// TIA Portal V21 export
FUNCTION "ANALOG" : Void   // FC9, LAD
{ S7_Optimized_Access := 'TRUE' }
// stored: SetENOAutomatically false
   VAR_TEMP
      DOOR1_P : Real;
      DOOR2_P : Real;
      CHAMBER_P : Real;
      JACKET_P : Real;
      NOM : Real;
      TEMP1 : Real;
   END_VAR
   VAR_TEMP   // added for the SCL form of the ladder/FBD networks
      _w1 : Bool;
      _w2 : Bool;
      _w3 : Bool;
   END_VAR
BEGIN

REGION Network 1: TEMPERATURE RTD
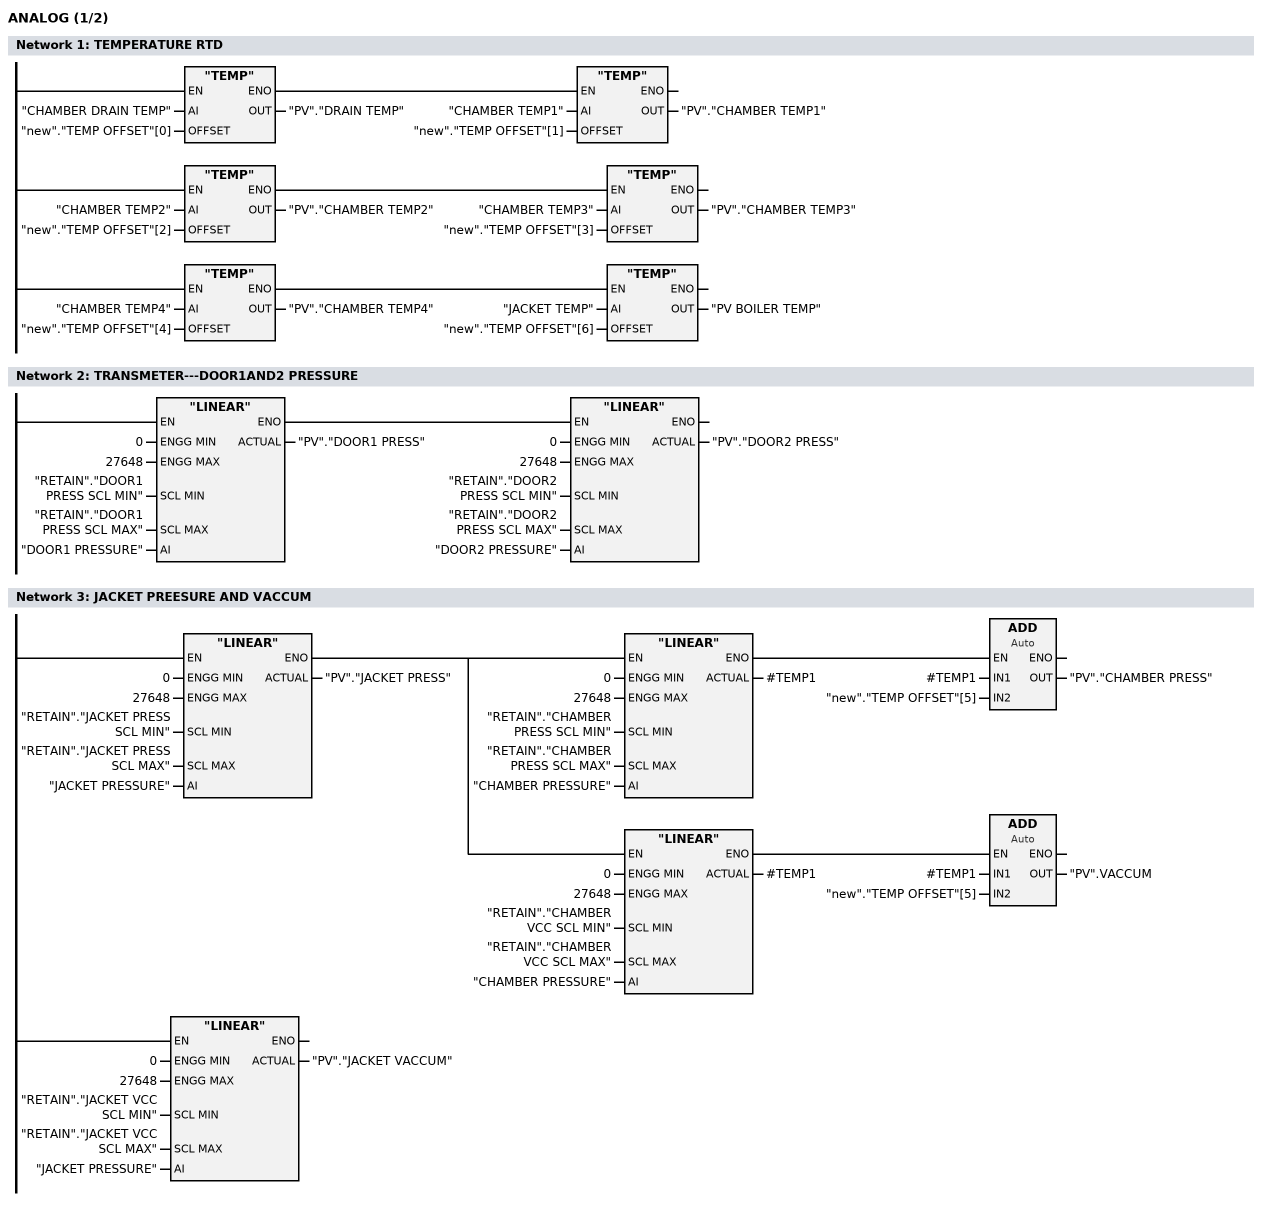
   RUNG wire#powerrail
      "TEMP"(AI := "CHAMBER DRAIN TEMP", OFFSET := "new"."TEMP OFFSET"[0], OUT => "PV"."DRAIN TEMP")
      "TEMP"(AI := "CHAMBER TEMP1", OFFSET := "new"."TEMP OFFSET"[1], OUT => "PV"."CHAMBER TEMP1")
   END_RUNG
   RUNG wire#powerrail
      "TEMP"(AI := "CHAMBER TEMP2", OFFSET := "new"."TEMP OFFSET"[2], OUT => "PV"."CHAMBER TEMP2")
      "TEMP"(AI := "CHAMBER TEMP3", OFFSET := "new"."TEMP OFFSET"[3], OUT => "PV"."CHAMBER TEMP3")
   END_RUNG
   RUNG wire#powerrail
      "TEMP"(AI := "CHAMBER TEMP4", OFFSET := "new"."TEMP OFFSET"[4], OUT => "PV"."CHAMBER TEMP4")
      "TEMP"(AI := "JACKET TEMP", OFFSET := "new"."TEMP OFFSET"[6], OUT => "PV BOILER TEMP")
   END_RUNG
   // the same network as SCL:
   "TEMP"(AI := "CHAMBER DRAIN TEMP", OFFSET := "new"."TEMP OFFSET"[0], OUT => "PV"."DRAIN TEMP", ENO => #_w1);
   IF #_w1 THEN
       "TEMP"(AI := "CHAMBER TEMP1", OFFSET := "new"."TEMP OFFSET"[1], OUT => "PV"."CHAMBER TEMP1");
   END_IF;
   "TEMP"(AI := "CHAMBER TEMP2", OFFSET := "new"."TEMP OFFSET"[2], OUT => "PV"."CHAMBER TEMP2", ENO => #_w2);
   IF #_w2 THEN
       "TEMP"(AI := "CHAMBER TEMP3", OFFSET := "new"."TEMP OFFSET"[3], OUT => "PV"."CHAMBER TEMP3");
   END_IF;
   "TEMP"(AI := "CHAMBER TEMP4", OFFSET := "new"."TEMP OFFSET"[4], OUT => "PV"."CHAMBER TEMP4", ENO => #_w3);
   IF #_w3 THEN
       "TEMP"(AI := "JACKET TEMP", OFFSET := "new"."TEMP OFFSET"[6], OUT => "PV BOILER TEMP");
   END_IF;
END_REGION

REGION Network 2: TRANSMETER---DOOR1AND2 PRESSURE
   RUNG wire#powerrail
      "LINEAR"("ENGG MIN" := 0, "ENGG MAX" := 27648, "SCL MIN" := "RETAIN"."DOOR1 PRESS SCL MIN", "SCL MAX" := "RETAIN"."DOOR1 PRESS SCL MAX", AI := "DOOR1 PRESSURE", ACTUAL => "PV"."DOOR1 PRESS")
      "LINEAR"("ENGG MIN" := 0, "ENGG MAX" := 27648, "SCL MIN" := "RETAIN"."DOOR2 PRESS SCL MIN", "SCL MAX" := "RETAIN"."DOOR2 PRESS SCL MAX", AI := "DOOR2 PRESSURE", ACTUAL => "PV"."DOOR2 PRESS")
   END_RUNG
   // the same network as SCL:
   "LINEAR"("ENGG MIN" := 0,
            "ENGG MAX" := 27648,
            "SCL MIN" := "RETAIN"."DOOR1 PRESS SCL MIN",
            "SCL MAX" := "RETAIN"."DOOR1 PRESS SCL MAX",
            AI := "DOOR1 PRESSURE",
            ACTUAL => "PV"."DOOR1 PRESS",
            ENO => #_w1);
   IF #_w1 THEN
       "LINEAR"("ENGG MIN" := 0,
                "ENGG MAX" := 27648,
                "SCL MIN" := "RETAIN"."DOOR2 PRESS SCL MIN",
                "SCL MAX" := "RETAIN"."DOOR2 PRESS SCL MAX",
                AI := "DOOR2 PRESSURE",
                ACTUAL => "PV"."DOOR2 PRESS");
   END_IF;
END_REGION

REGION Network 3: JACKET PREESURE AND VACCUM
   RUNG wire#powerrail
      "LINEAR"("ENGG MIN" := 0, "ENGG MAX" := 27648, "SCL MIN" := "RETAIN"."JACKET PRESS SCL MIN", "SCL MAX" := "RETAIN"."JACKET PRESS SCL MAX", AI := "JACKET PRESSURE", ACTUAL => "PV"."JACKET PRESS")
      wire#w1
      "LINEAR"("ENGG MIN" := 0, "ENGG MAX" := 27648, "SCL MIN" := "RETAIN"."CHAMBER PRESS SCL MIN", "SCL MAX" := "RETAIN"."CHAMBER PRESS SCL MAX", AI := "CHAMBER PRESSURE", ACTUAL => #TEMP1)
      Add(in1 := #TEMP1, in2 := "new"."TEMP OFFSET"[5], out => "PV"."CHAMBER PRESS")
   END_RUNG
   RUNG wire#w1
      "LINEAR"("ENGG MIN" := 0, "ENGG MAX" := 27648, "SCL MIN" := "RETAIN"."CHAMBER VCC SCL MIN", "SCL MAX" := "RETAIN"."CHAMBER VCC SCL MAX", AI := "CHAMBER PRESSURE", ACTUAL => #TEMP1)
      Add(in1 := #TEMP1, in2 := "new"."TEMP OFFSET"[5], out => "PV".VACCUM)
   END_RUNG
   RUNG wire#powerrail
      "LINEAR"("ENGG MIN" := 0, "ENGG MAX" := 27648, "SCL MIN" := "RETAIN"."JACKET VCC SCL MIN", "SCL MAX" := "RETAIN"."JACKET VCC SCL MAX", AI := "JACKET PRESSURE", ACTUAL => "PV"."JACKET VACCUM")
   END_RUNG
   // the same network as SCL:
   "LINEAR"("ENGG MIN" := 0,
            "ENGG MAX" := 27648,
            "SCL MIN" := "RETAIN"."JACKET PRESS SCL MIN",
            "SCL MAX" := "RETAIN"."JACKET PRESS SCL MAX",
            AI := "JACKET PRESSURE",
            ACTUAL => "PV"."JACKET PRESS",
            ENO => #_w1);
   "LINEAR"(EN := #_w1,
            "ENGG MIN" := 0,
            "ENGG MAX" := 27648,
            "SCL MIN" := "RETAIN"."CHAMBER PRESS SCL MIN",
            "SCL MAX" := "RETAIN"."CHAMBER PRESS SCL MAX",
            AI := "CHAMBER PRESSURE",
            ACTUAL => #TEMP1,
            ENO => #_w2);
   IF #_w2 THEN "PV"."CHAMBER PRESS" := #TEMP1 + "new"."TEMP OFFSET"[5]; END_IF;
   "LINEAR"(EN := #_w1,
            "ENGG MIN" := 0,
            "ENGG MAX" := 27648,
            "SCL MIN" := "RETAIN"."CHAMBER VCC SCL MIN",
            "SCL MAX" := "RETAIN"."CHAMBER VCC SCL MAX",
            AI := "CHAMBER PRESSURE",
            ACTUAL => #TEMP1,
            ENO => #_w3);
   IF #_w3 THEN "PV".VACCUM := #TEMP1 + "new"."TEMP OFFSET"[5]; END_IF;
   "LINEAR"("ENGG MIN" := 0,
            "ENGG MAX" := 27648,
            "SCL MIN" := "RETAIN"."JACKET VCC SCL MIN",
            "SCL MAX" := "RETAIN"."JACKET VCC SCL MAX",
            AI := "JACKET PRESSURE",
            ACTUAL => "PV"."JACKET VACCUM");
END_REGION

REGION Network 4: DOOR1AND 2 VACCUM
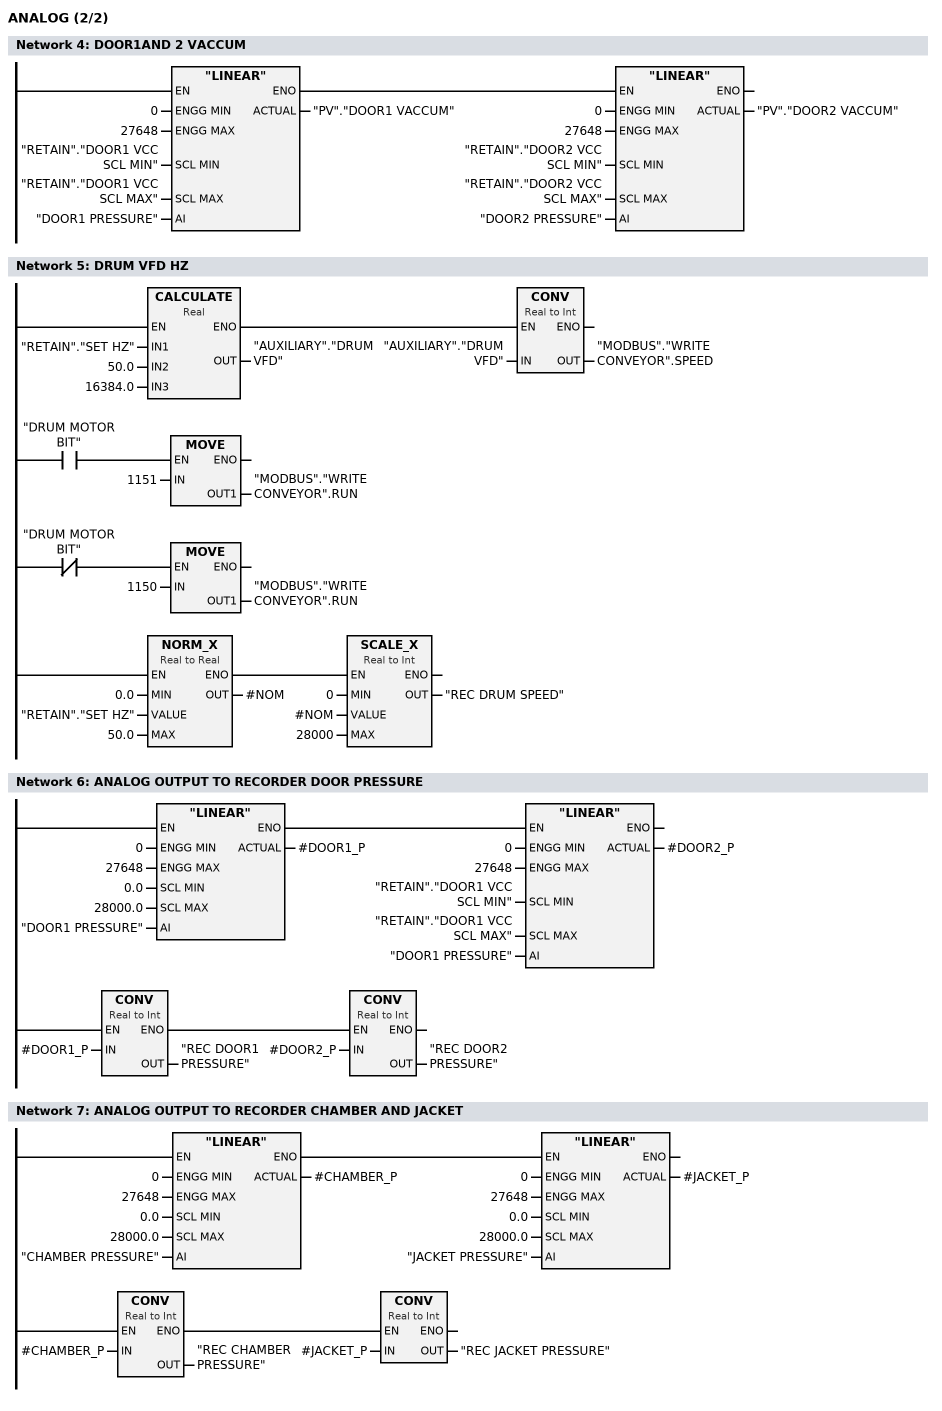
   RUNG wire#powerrail
      "LINEAR"("ENGG MIN" := 0, "ENGG MAX" := 27648, "SCL MIN" := "RETAIN"."DOOR1 VCC SCL MIN", "SCL MAX" := "RETAIN"."DOOR1 VCC SCL MAX", AI := "DOOR1 PRESSURE", ACTUAL => "PV"."DOOR1 VACCUM")
      "LINEAR"("ENGG MIN" := 0, "ENGG MAX" := 27648, "SCL MIN" := "RETAIN"."DOOR2 VCC SCL MIN", "SCL MAX" := "RETAIN"."DOOR2 VCC SCL MAX", AI := "DOOR2 PRESSURE", ACTUAL => "PV"."DOOR2 VACCUM")
   END_RUNG
   // the same network as SCL:
   "LINEAR"("ENGG MIN" := 0,
            "ENGG MAX" := 27648,
            "SCL MIN" := "RETAIN"."DOOR1 VCC SCL MIN",
            "SCL MAX" := "RETAIN"."DOOR1 VCC SCL MAX",
            AI := "DOOR1 PRESSURE",
            ACTUAL => "PV"."DOOR1 VACCUM",
            ENO => #_w1);
   IF #_w1 THEN
       "LINEAR"("ENGG MIN" := 0,
                "ENGG MAX" := 27648,
                "SCL MIN" := "RETAIN"."DOOR2 VCC SCL MIN",
                "SCL MAX" := "RETAIN"."DOOR2 VCC SCL MAX",
                AI := "DOOR2 PRESSURE",
                ACTUAL => "PV"."DOOR2 VACCUM");
   END_IF;
END_REGION

REGION Network 5: DRUM VFD HZ
   RUNG wire#powerrail
      { S7_Templates := "SrcType := Real"; S7_Expression := "(IN1/IN2)*IN3" } Calculate(in1 := "RETAIN"."SET HZ", in2 := 50.0, in3 := 16384.0, out => "AUXILIARY"."DRUM VFD")
      { S7_Templates := "[SrcType := Real, DestType := Int]" } Convert(in := "AUXILIARY"."DRUM VFD", out => "MODBUS"."WRITE CONVEYOR".SPEED)
   END_RUNG
   RUNG wire#powerrail
      Contact( "DRUM MOTOR BIT" )
      Move(in := 1151, out1 => "MODBUS"."WRITE CONVEYOR".RUN)
   END_RUNG
   RUNG wire#powerrail
      I_Contact( "DRUM MOTOR BIT" )
      Move(in := 1150, out1 => "MODBUS"."WRITE CONVEYOR".RUN)
   END_RUNG
   RUNG wire#powerrail
      { S7_Templates := "[SrcType := Real, DestType := Real]" } Normalize(min := 0.0, value := "RETAIN"."SET HZ", max := 50.0, out => #NOM)
      { S7_Templates := "[SrcType := Real, DestType := Int]" } Scale(min := 0, value := #NOM, max := 28000, out => "REC DRUM SPEED")
   END_RUNG
   // the same network as SCL:
   "AUXILIARY"."DRUM VFD" := ("RETAIN"."SET HZ"/50.0)*16384.0;
   "MODBUS"."WRITE CONVEYOR".SPEED := REAL_TO_INT("AUXILIARY"."DRUM VFD");
   IF "DRUM MOTOR BIT" THEN "MODBUS"."WRITE CONVEYOR".RUN := 1151; END_IF;
   IF NOT "DRUM MOTOR BIT" THEN "MODBUS"."WRITE CONVEYOR".RUN := 1150; END_IF;
   #NOM := NORM_X(MIN := 0.0, VALUE := "RETAIN"."SET HZ", MAX := 50.0);
   "REC DRUM SPEED" := SCALE_X(MIN := 0, VALUE := #NOM, MAX := 28000);
END_REGION

REGION Network 6: ANALOG OUTPUT TO RECORDER DOOR PRESSURE
   RUNG wire#powerrail
      "LINEAR"("ENGG MIN" := 0, "ENGG MAX" := 27648, "SCL MIN" := 0.0, "SCL MAX" := 28000.0, AI := "DOOR1 PRESSURE", ACTUAL => #DOOR1_P)
      "LINEAR"("ENGG MIN" := 0, "ENGG MAX" := 27648, "SCL MIN" := "RETAIN"."DOOR1 VCC SCL MIN", "SCL MAX" := "RETAIN"."DOOR1 VCC SCL MAX", AI := "DOOR1 PRESSURE", ACTUAL => #DOOR2_P)
   END_RUNG
   RUNG wire#powerrail
      { S7_Templates := "[SrcType := Real, DestType := Int]" } Convert(in := #DOOR1_P, out => "REC DOOR1 PRESSURE")
      { S7_Templates := "[SrcType := Real, DestType := Int]" } Convert(in := #DOOR2_P, out => "REC DOOR2 PRESSURE")
   END_RUNG
   // the same network as SCL:
   "LINEAR"("ENGG MIN" := 0,
            "ENGG MAX" := 27648,
            "SCL MIN" := 0.0,
            "SCL MAX" := 28000.0,
            AI := "DOOR1 PRESSURE",
            ACTUAL => #DOOR1_P,
            ENO => #_w1);
   IF #_w1 THEN
       "LINEAR"("ENGG MIN" := 0,
                "ENGG MAX" := 27648,
                "SCL MIN" := "RETAIN"."DOOR1 VCC SCL MIN",
                "SCL MAX" := "RETAIN"."DOOR1 VCC SCL MAX",
                AI := "DOOR1 PRESSURE",
                ACTUAL => #DOOR2_P);
   END_IF;
   "REC DOOR1 PRESSURE" := REAL_TO_INT(#DOOR1_P);
   "REC DOOR2 PRESSURE" := REAL_TO_INT(#DOOR2_P);
END_REGION

REGION Network 7: ANALOG OUTPUT TO RECORDER CHAMBER AND JACKET
   RUNG wire#powerrail
      "LINEAR"("ENGG MIN" := 0, "ENGG MAX" := 27648, "SCL MIN" := 0.0, "SCL MAX" := 28000.0, AI := "CHAMBER PRESSURE", ACTUAL => #CHAMBER_P)
      "LINEAR"("ENGG MIN" := 0, "ENGG MAX" := 27648, "SCL MIN" := 0.0, "SCL MAX" := 28000.0, AI := "JACKET PRESSURE", ACTUAL => #JACKET_P)
   END_RUNG
   RUNG wire#powerrail
      { S7_Templates := "[SrcType := Real, DestType := Int]" } Convert(in := #CHAMBER_P, out => "REC CHAMBER PRESSURE")
      { S7_Templates := "[SrcType := Real, DestType := Int]" } Convert(in := #JACKET_P, out => "REC JACKET PRESSURE")
   END_RUNG
   // the same network as SCL:
   "LINEAR"("ENGG MIN" := 0,
            "ENGG MAX" := 27648,
            "SCL MIN" := 0.0,
            "SCL MAX" := 28000.0,
            AI := "CHAMBER PRESSURE",
            ACTUAL => #CHAMBER_P,
            ENO => #_w1);
   IF #_w1 THEN
       "LINEAR"("ENGG MIN" := 0,
                "ENGG MAX" := 27648,
                "SCL MIN" := 0.0,
                "SCL MAX" := 28000.0,
                AI := "JACKET PRESSURE",
                ACTUAL => #JACKET_P);
   END_IF;
   "REC CHAMBER PRESSURE" := REAL_TO_INT(#CHAMBER_P);
   "REC JACKET PRESSURE" := REAL_TO_INT(#JACKET_P);
END_REGION
END_FUNCTION
